FUNCTION F_DCTimestructToFileTime : ULINT
VAR_INPUT
	dtTimestamp: DCTIMESTRUCT;
END_VAR
VAR
	dcTime: T_DCTIME64;
END_VAR

dcTime:= DCTIMESTRUCT_TO_DCTIME64(dtTimestamp);
F_DCTimestructToFileTime:= F_AlyTimestampToFileTime(dcTime);

END_FUNCTION

(* stored: POU F_DCTimestructToFileTime: Id 781619b6-f88f-406c-aa85-d030aa8dbc6e, SpecialFunc None *)
